// TIA Portal V19 export
DATA_BLOCK "DB_Panel_LZ"   // DB81
{ S7_Optimized_Access := 'FALSE' }
AUTHOR : KHE_RE
NAME : DB_LADUN
VERSION : 2.0
// stored: AutoNumber false
   VAR RETAIN
      Anz : Int := 0;   // wird aus DB1 übernommen
      Offset : Int := 20;   // * Beginn Daten
      Length : Int := 36;   // * Länge Daten
      resB6 : Byte := 16#00;
      resB7 : Byte := 16#00;
      resD8 : DWord := 16#0000_0000;
      resD12 : DWord := 16#0000_0000;
      resD16 : DWord := 16#0000_0000;
      Becken : Array[1..20] of Struct   // * Feldlänge anpassen
         Dosi_Int : DInt;   // Abstand zw. 2 Dosierungen (Sollw.)
         Dosi_Zaehl : DInt;   // Ladung nach letzter Dosierung (Istw.)
         Rest_Zaehl1 : DInt;
         Ladu_Zaehl1 : DInt;   // kont. Ladungszähler 1 (Soll/Istw.)
         Ladu_Zaehl2 : DInt;   // kont. Ladungszähler 2 (Soll/Istw.)
         Ladu_Zaehl3 : DInt;   // kont. Ladungszähler 3 (Soll/Istw.)
         Ladu_Zaehl4 : DInt;   // kont. Ladungszähler 4 (Soll/Istw.)
         Ladu_Zaehl5 : DInt;   // kont. Ladungszähler 5 (Soll/Istw.)
         Ladu_Zaehl6 : DInt;   // kont. Ladungszähler 6 (Soll/Istw.)
      END_STRUCT;
   END_VAR
BEGIN
   Becken[1..20].Dosi_Int := 1000;
   Becken[1..20].Dosi_Zaehl := 0;
   Becken[1..20].Rest_Zaehl1 := 0;
   Becken[1..20].Ladu_Zaehl1 := 0;
   Becken[1..20].Ladu_Zaehl2 := 0;
   Becken[1..20].Ladu_Zaehl3 := 0;
   Becken[1..20].Ladu_Zaehl4 := 0;
   Becken[1..20].Ladu_Zaehl5 := 0;
   Becken[1..20].Ladu_Zaehl6 := 0;
END_DATA_BLOCK
